(* PLC project SafeLOGIC-1, BrAutomation SafeDESIGNER  5.15.0.0 *)
(* stored: companyURL http://www.br-automation.com, creationDateTime Wed Sep 14 14:43:20 2022 *)

PROGRAM ReleaseOutput

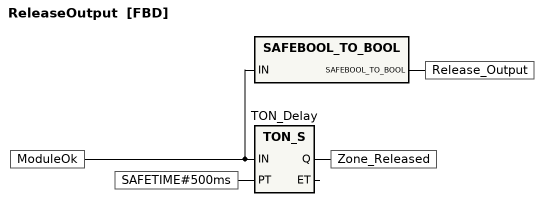
(* FBD diagram, written out as Structured Text *)
Release_Output := SAFEBOOL_TO_BOOL(ModuleOk);
TON_Delay(IN := ModuleOk, PT := SAFETIME#500ms);
Zone_Released := TON_Delay.Q;
END_PROGRAM
